VAR_GLOBAL
    // Semantic version in machine-readable format.
    // Update it and commit it immediatly before setting a tag
    nVersionMajor: UINT := 2; // Major Version
    nVersionMinor: UINT := 2; // Minor Version
    nVersionPatch: UINT := 0; // Patch level
    astAxes: ARRAY [1..GVL_APP.nAXIS_NUM] OF ST_AxisStruct; //Array of ST_AxisStruct for holding axis parameters and controls
    astPneumaticAxes: ARRAY [1..GVL_APP.nPNEUMATIC_AXIS_NUM] OF ST_PneumaticAxisStruct; //Array of ST_PneumaticAxisStruct for holding pneumatic axis parameters and controls
    iAxis: UINT; //Index for for loops while going through axes
	iSafety: UINT; //Index for loops while going through safety devices
    iGroup: INT;
	iPneumaticAxis: UINT := 1; //Index for for loops while going through pneumatic axes
    fbGetCurTaskIndex: GETCURTASKINDEX;
    bLocalMode: BOOL;
	astAxesPersistent: ARRAY [1..GVL_APP.nAXIS_NUM] OF ST_AxisPersistent;
	astAxesGroup: ARRAY [1..GVL_APP.nAXIS_GROUPS_NUM] OF ST_AxisGroupStruct;
	iAxesGroupIndex : INT;
END_VAR

VAR_GLOBAL CONSTANT
    nMAX_AXIS_NAME: UINT := 32;
    nMAX_AXIS_GROUP_NAME: UINT := 32;
	nMAX_AXES_PER_GROUP: INT := 9;	nMAX_SAFETY_NAME: UINT := 32;
	nMAX_LOCATION_NAME: UINT := 32;
END_VAR

(* stored: Version 1.1.0.1, ProductVersion 3.1.4026.18
   GVL GVL: Id {913e21aa-a47e-444c-bfce-679b16c0434b} *)
